// TIA Portal V18 export
TYPE "LGasp_TypeData_toERP"
// stored: IsFailsafeCompliant false
   STRUCT
      ID_inizio_ODL : DInt;   // ID associato a evento "inizio ODL"
      ID_fine_ODL : DInt;   // ID associato a evento "fine ODL"
      ID_fine_pacco : DInt;   // ID associato a evento "fine pacco"
      ID_pezzo_tagliato : DInt;   // ID associato a evento "pezzo tagliato"
      ID_articolo_terminato : DInt;   // ID associato a evento "articolo terminato"
      lunghezza_pezzo_tagliato : LReal;   // [mm] Lunghezza associata a evento "pezzo tagliato"
      lunghezza_articolo_terminato : LReal;   // [mm] Lunghezza associata a evento "articolo teminato"
      coilsetup : Array[1..4] of "LGasp_TypeCoil_fromERP";
   END_STRUCT;
END_TYPE
